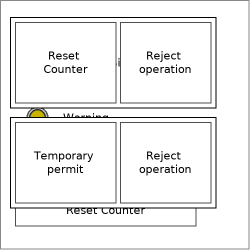
VISUALIZATION vMachineCycleCounter_V2  // 250x250
VAR_IN_OUT
	fb			: fbMachineCycleCounter;
END_VAR
    Rectangle (15,195 181x31), "Reset Counter", input disabled if: NOT fb.bBlocked
        OnMouseClick: toggle fb.bResetAqusitton
    Rectangle (15,160 181x31), "Temporary permit", input disabled if: NOT fb.bBlocked
        OnMouseClick: toggle fb.bTempolaryPermit
    Lamp1 (25,105 25x25), variable: fb.bWarning, style: Lamp-Lamp1-Yellow
    Rectangle (60,105 160x26), "Warning"
    Rectangle (60,135 106x25), "Limit exceeded"
    Lamp1 (25,135 25x25), variable: fb.bError, style: Lamp-Lamp1-Yellow
    Rectangle (10,17 206x91), invisible if: fb.bResetAqusitton
    Rectangle (10,117 206x91), invisible if: fb.bTempolaryPermit
    Rectangle (26,71 160x26), "Loged User: %s", text variable: fb.sUserName
    Rectangle (26,50 160x26), "Cover Cycles: %i", text variable: fb.iOperationCalcHMI
    Rectangle (26,27 160x26), "Total: %i", text variable: fb.iCyclesCalcHMI
    Rectangle (15,22 101x81), "Reset Counter", invisible if: fb.bResetAqusitton
        OnMouseClick: toggle fb.bResetAqusitton
        OnMouseClick: toggle fb.bReset
    Rectangle (120,22 91x81), "Reject operation", invisible if: fb.bResetAqusitton
        OnMouseClick: toggle fb.bResetAqusitton
    Rectangle (120,122 91x81), "Reject operation", invisible if: fb.bTempolaryPermit
        OnMouseClick: toggle fb.bTempolaryPermit
    Rectangle (15,122 101x81), "Temporary permit", invisible if: fb.bTempolaryPermit
        OnMouseClick: toggle fb.bClear
        OnMouseClick: toggle fb.bTempolaryPermit
END_VISUALIZATION

(* stored: Version 1.1.0.1, ProductVersion 3.1.4024.13
   Visu vMachineCycleCounter_V2: Id {6533fb15-f659-4d22-a383-c0b564d79c81} *)
